FUNCTION PercentToAnalog : INT
VAR_INPUT
	TargetValue : DINT; // 0-100%
END_VAR

PercentToAnalog := TO_INT(32767 * TargetValue / 100);

END_FUNCTION

(* stored: Version 1.1.0.1, ProductVersion 3.1.4026.18
   POU PercentToAnalog: Id {0784c406-0ba0-0383-21cb-aa47f0a84b53}, SpecialFunc None *)
